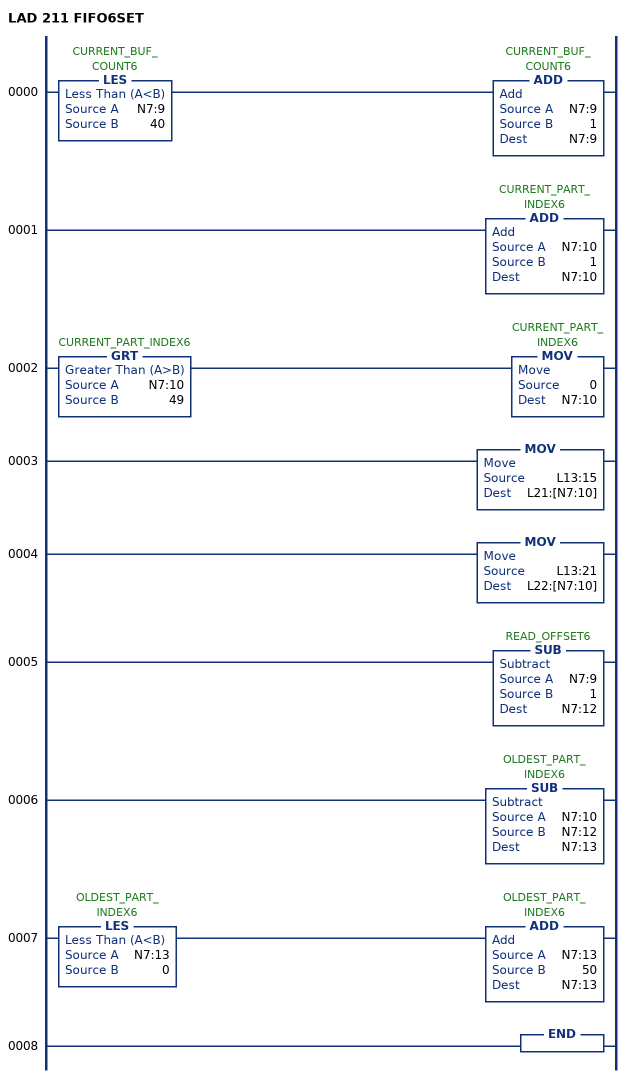
% Rung: 0 %
SOR LES N7:9 40 ADD N7:9 1 N7:9 EOR
%   N7:9  CURRENT_BUF_COUNT6 %
% Rung: 1 %
SOR ADD N7:10 1 N7:10 EOR
%   N7:10  CURRENT_PART_INDEX6 %
% Rung: 2 %
SOR GRT N7:10 49 MOV 0 N7:10 EOR
%   N7:10  CURRENT_PART_INDEX6 %
% Rung: 3 %
SOR MOV L13:15 L21:[N7:10] EOR
%   L13:15  TOP_TIME %
%   N7:10  CURRENT_PART_INDEX6 %
% Rung: 4 %
SOR MOV L13:21 L22:[N7:10] EOR
%   L13:21  TOP_POSITION %
%   N7:10  CURRENT_PART_INDEX6 %
% Rung: 5 %
SOR SUB N7:9 1 N7:12 EOR
%   N7:9  CURRENT_BUF_COUNT6 %
%   N7:12  READ_OFFSET6 %
% Rung: 6 %
SOR SUB N7:10 N7:12 N7:13 EOR
%   N7:10  CURRENT_PART_INDEX6 %
%   N7:12  READ_OFFSET6 %
%   N7:13  OLDEST_PART_INDEX6 %
% Rung: 7 %
SOR LES N7:13 0 ADD N7:13 50 N7:13 EOR
%   N7:13  OLDEST_PART_INDEX6 %
% Rung: 8 %
SOR END EOR

LADDER 212 "FIFO6GET"
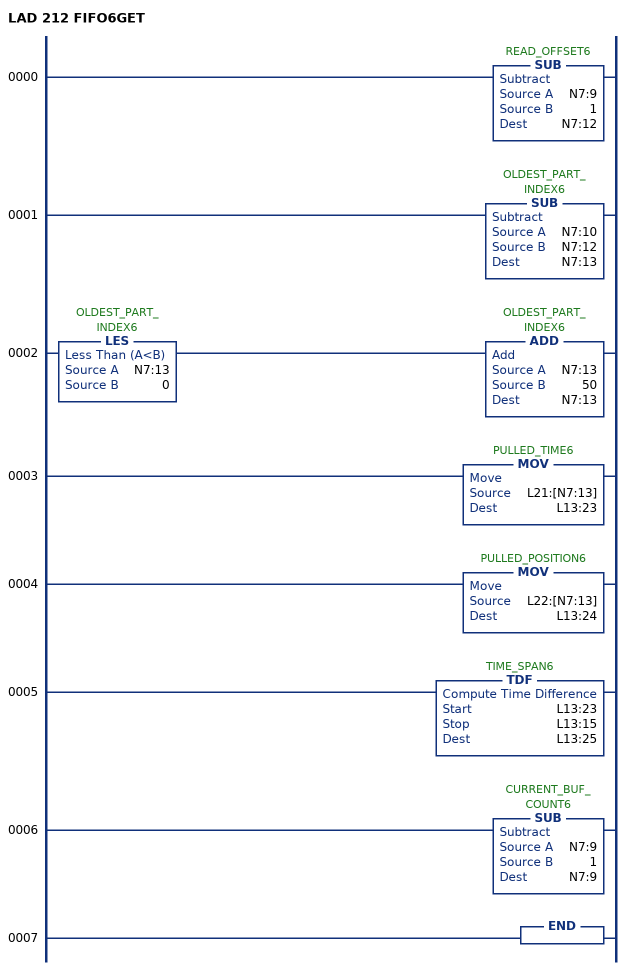
% Rung: 0 %
SOR SUB N7:9 1 N7:12 EOR
%   N7:9  CURRENT_BUF_COUNT6 %
%   N7:12  READ_OFFSET6 %
% Rung: 1 %
SOR SUB N7:10 N7:12 N7:13 EOR
%   N7:10  CURRENT_PART_INDEX6 %
%   N7:12  READ_OFFSET6 %
%   N7:13  OLDEST_PART_INDEX6 %
% Rung: 2 %
SOR LES N7:13 0 ADD N7:13 50 N7:13 EOR
%   N7:13  OLDEST_PART_INDEX6 %
% Rung: 3 %
SOR MOV L21:[N7:13] L13:23 EOR
%   N7:13  OLDEST_PART_INDEX6 %
%   L13:23  PULLED_TIME6 %
% Rung: 4 %
SOR MOV L22:[N7:13] L13:24 EOR
%   N7:13  OLDEST_PART_INDEX6 %
%   L13:24  PULLED_POSITION6 %
% Rung: 5 %
SOR TDF L13:23 L13:15 L13:25 EOR
%   L13:23  PULLED_TIME6 %
%   L13:15  TOP_TIME %
%   L13:25  TIME_SPAN6 %
% Rung: 6 %
SOR SUB N7:9 1 N7:9 EOR
%   N7:9  CURRENT_BUF_COUNT6 %
% Rung: 7 %
SOR END EOR

LADDER 213 "INSDATA6"
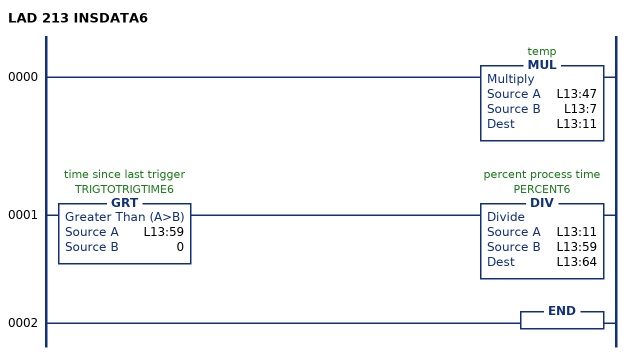
% Rung: 0 %
SOR MUL L13:47 L13:7 L13:11 EOR
%   L13:47  PROCESSTIME6  "process 6 time" %
%   L13:7  PERCENT_MULTIPLYER %
%   L13:11  "temp" %
% Rung: 1 %
SOR GRT L13:59 0 DIV L13:11 L13:59 L13:64 EOR
%   L13:59  TRIGTOTRIGTIME6  "time since last trigger" %
%   L13:11  "temp" %
%   L13:64  PERCENT6  "percent process time" %
% Rung: 2 %
SOR END EOR

LADDER 214 "TESTFAULT6"
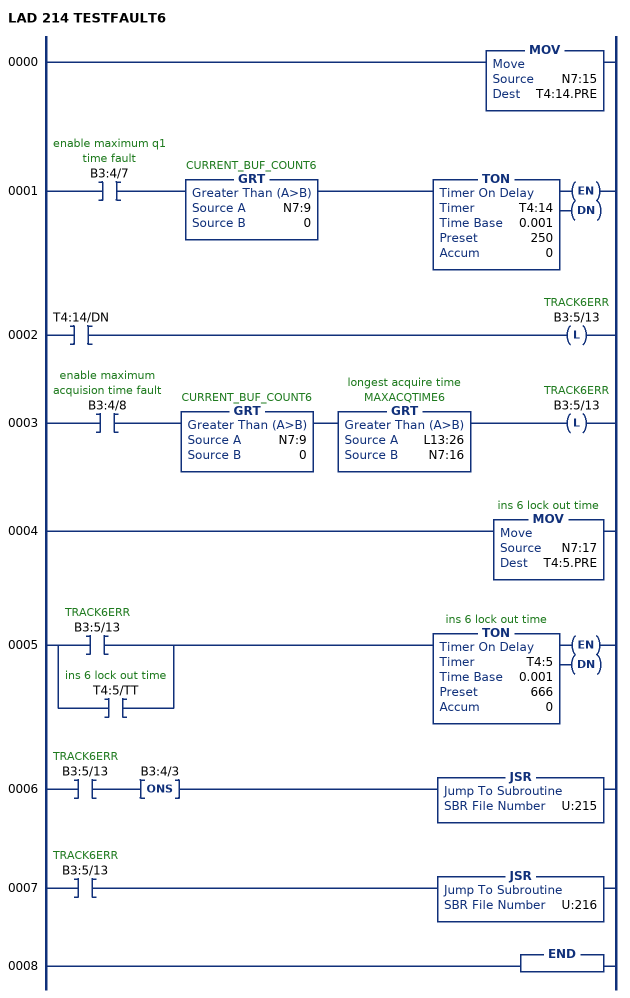
% Rung: 0 %
SOR MOV N7:15 T4:14.PRE EOR
%   N7:15  "max allowed ms time for q to be above 1 if safe fault is used" %
% Rung: 1 %
SOR XIC B3:4/7 GRT N7:9 0 TON T4:14 0.001 250 0 EOR
%   B3:4/7  "enable maximum q1 time fault" %
%   N7:9  CURRENT_BUF_COUNT6 %
% Rung: 2 %
SOR XIC T4:14/DN OTL B3:5/13 EOR
%   B3:5/13  TRACK6ERR %
% Rung: 3 %
SOR XIC B3:4/8 GRT N7:9 0 GRT L13:26 N7:16 OTL B3:5/13 EOR
%   B3:4/8  "enable maximum acquision time fault" %
%   N7:9  CURRENT_BUF_COUNT6 %
%   L13:26  MAXACQTIME6  "longest acquire time" %
%   N7:16  ACQUIRE_TIME_LIMIT  "maximum of the longest acquire time allowed if maximum acquire time fault is enabled" %
%   B3:5/13  TRACK6ERR %
% Rung: 4 %
SOR MOV N7:17 T4:5.PRE EOR
%   N7:17  "ms time setting to lock out inspection to give all pending images a chance to clear" %
%   T4:5  "ins 6 lock out time" %
% Rung: 5 %
SOR BST XIC B3:5/13 NXB XIC T4:5/TT BND TON T4:5 0.001 666 0 EOR
%   B3:5/13  TRACK6ERR %
%   T4:5  "ins 6 lock out time" %
% Rung: 6 %
SOR XIC B3:5/13 ONS B3:4/3 JSR U:215 EOR
%   B3:5/13  TRACK6ERR %
% Rung: 7 %
SOR XIC B3:5/13 JSR U:216 EOR
%   B3:5/13  TRACK6ERR %
% Rung: 8 %
SOR END EOR

LADDER 215 "INS6FIX1"
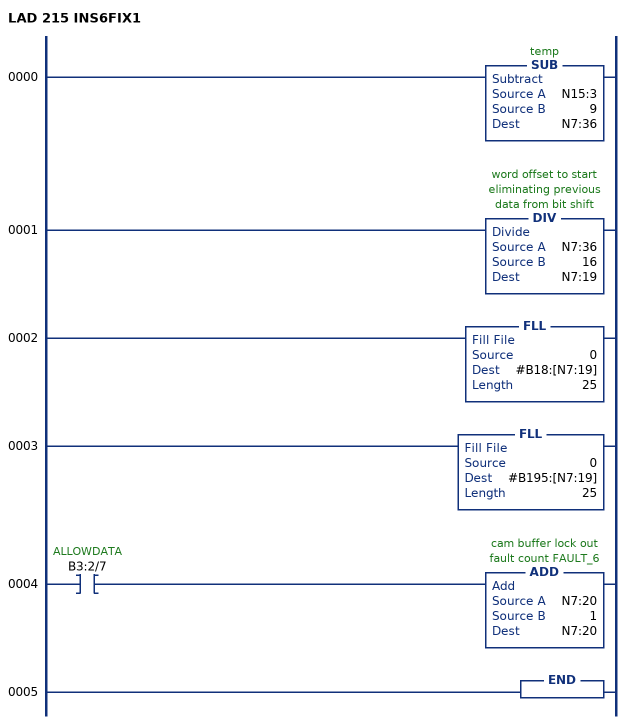
% Rung: 0 %
SOR SUB N15:3 9 N7:36 EOR
%   N15:3  INS_6_TRIG_LOC %
%   N7:36  "temp" %
% Rung: 1 %
SOR DIV N7:36 16 N7:19 EOR
%   N7:36  "temp" %
%   N7:19  "word offset to start eliminating previous data from bit shift" %
% Rung: 2 %
SOR FLL 0 #B18:[N7:19] 25 EOR
%   N7:19  "word offset to start eliminating previous data from bit shift" %
% Rung: 3 %
SOR FLL 0 #B195:[N7:19] 25 EOR
%   N7:19  "word offset to start eliminating previous data from bit shift" %
% Rung: 4 %
SOR XIC B3:2/7 ADD N7:20 1 N7:20 EOR
%   B3:2/7  ALLOWDATA %
%   N7:20  FAULT_6  "cam buffer lock out fault count" %
% Rung: 5 %
SOR END EOR

LADDER 216 "INS6FIX2"
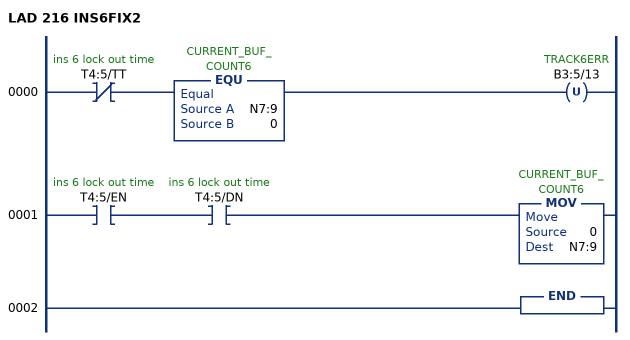
% Rung: 0 %
SOR XIO T4:5/TT EQU N7:9 0 OTU B3:5/13 EOR
%   T4:5  "ins 6 lock out time" %
%   N7:9  CURRENT_BUF_COUNT6 %
%   B3:5/13  TRACK6ERR %
% Rung: 1 %
SOR XIC T4:5/EN XIC T4:5/DN MOV 0 N7:9 EOR
%   T4:5  "ins 6 lock out time" %
%   N7:9  CURRENT_BUF_COUNT6 %
% Rung: 2 %
SOR END EOR

LADDER 218 "INS7"
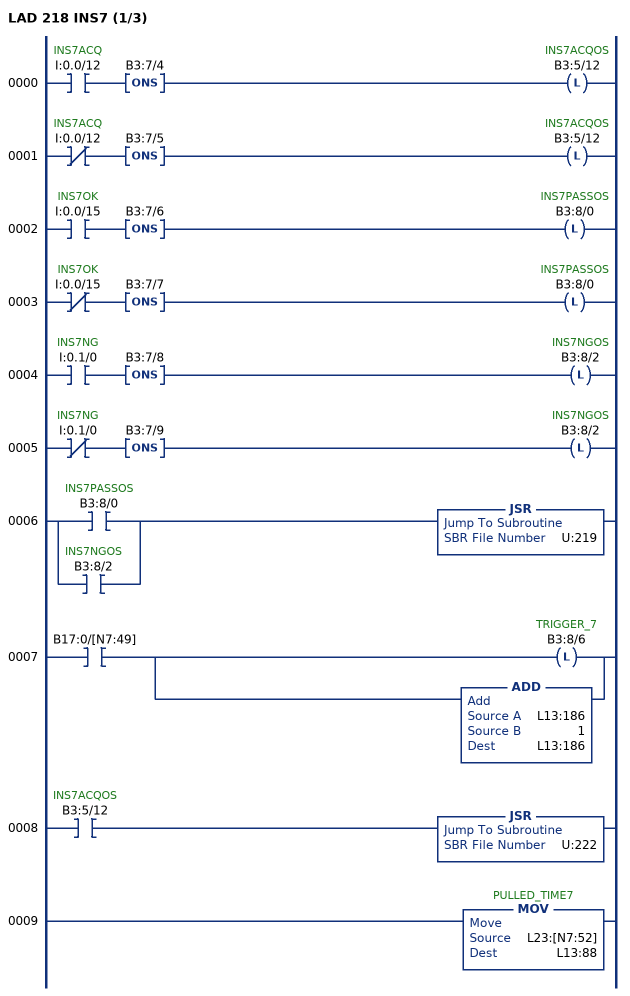
% Rung: 0 %
SOR XIC I:0.0/12 ONS B3:7/4 OTL B3:5/12 EOR
%   I:0.0/12  INS7ACQ %
%   B3:5/12  INS7ACQOS %
% Rung: 1 %
SOR XIO I:0.0/12 ONS B3:7/5 OTL B3:5/12 EOR
%   I:0.0/12  INS7ACQ %
%   B3:5/12  INS7ACQOS %
% Rung: 2 %
SOR XIC I:0.0/15 ONS B3:7/6 OTL B3:8/0 EOR
%   I:0.0/15  INS7OK %
%   B3:8/0  INS7PASSOS %
% Rung: 3 %
SOR XIO I:0.0/15 ONS B3:7/7 OTL B3:8/0 EOR
%   I:0.0/15  INS7OK %
%   B3:8/0  INS7PASSOS %
% Rung: 4 %
SOR XIC I:0.1/0 ONS B3:7/8 OTL B3:8/2 EOR
%   I:0.1/0  INS7NG %
%   B3:8/2  INS7NGOS %
% Rung: 5 %
SOR XIO I:0.1/0 ONS B3:7/9 OTL B3:8/2 EOR
%   I:0.1/0  INS7NG %
%   B3:8/2  INS7NGOS %
% Rung: 6 %
SOR BST XIC B3:8/0 NXB XIC B3:8/2 BND JSR U:219 EOR
%   B3:8/0  INS7PASSOS %
%   B3:8/2  INS7NGOS %
% Rung: 7 %
SOR XIC B17:0/[N7:49] BST OTL B3:8/6 NXB ADD L13:186 1 L13:186 BND EOR
%   B17:0  GOOD1 %
%   N7:49  INS_7_TRIG_LOC %
%   B3:8/6  TRIGGER_7 %
% Rung: 8 %
SOR XIC B3:5/12 JSR U:222 EOR
%   B3:5/12  INS7ACQOS %
% Rung: 9 %
SOR MOV L23:[N7:52] L13:88 EOR
%   N7:52  OLDEST_PART_INDEX7 %
%   L13:88  PULLED_TIME7 %

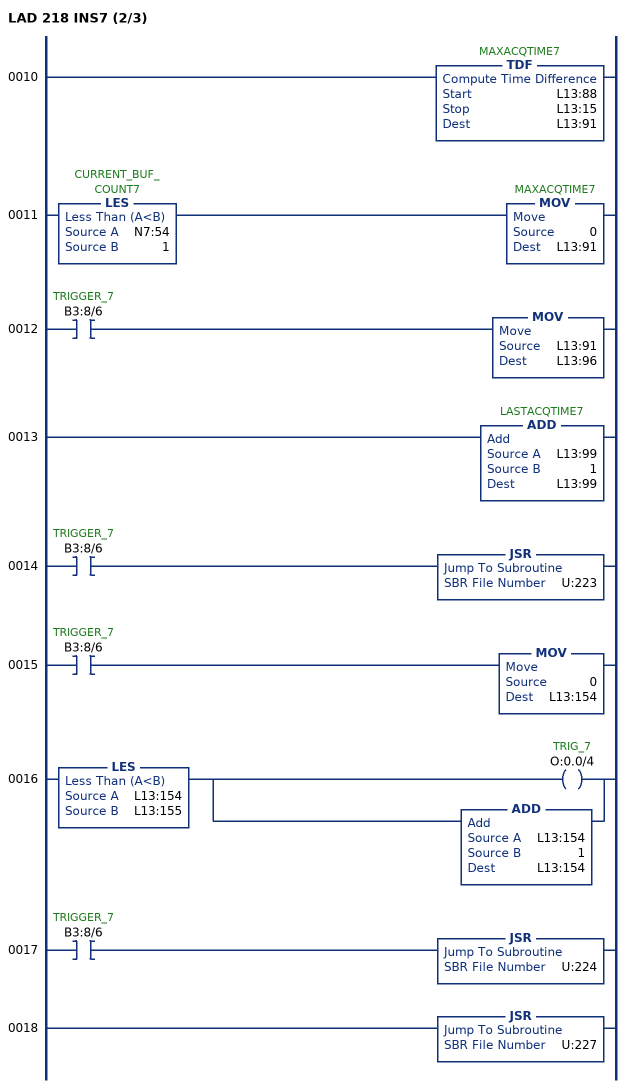
% Rung: 10 %
SOR TDF L13:88 L13:15 L13:91 EOR
%   L13:88  PULLED_TIME7 %
%   L13:15  TOP_TIME %
%   L13:91  MAXACQTIME7 %
% Rung: 11 %
SOR LES N7:54 1 MOV 0 L13:91 EOR
%   N7:54  CURRENT_BUF_COUNT7 %
%   L13:91  MAXACQTIME7 %
% Rung: 12 %
SOR XIC B3:8/6 MOV L13:91 L13:96 EOR
%   B3:8/6  TRIGGER_7 %
%   L13:91  MAXACQTIME7 %
% Rung: 13 %
SOR ADD L13:99 1 L13:99 EOR
%   L13:99  LASTACQTIME7 %
% Rung: 14 %
SOR XIC B3:8/6 JSR U:223 EOR
%   B3:8/6  TRIGGER_7 %
% Rung: 15 %
SOR XIC B3:8/6 MOV 0 L13:154 EOR
%   B3:8/6  TRIGGER_7 %
% Rung: 16 %
SOR LES L13:154 L13:155 BST OTE O:0.0/4 NXB ADD L13:154 1 L13:154 BND EOR
%   O:0.0/4  TRIG_7 %
% Rung: 17 %
SOR XIC B3:8/6 JSR U:224 EOR
%   B3:8/6  TRIGGER_7 %
% Rung: 18 %
SOR JSR U:227 EOR

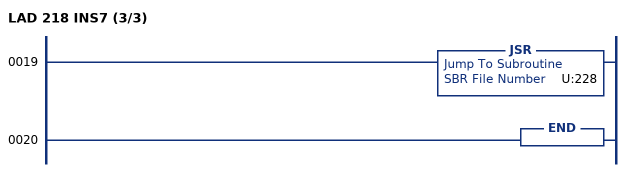
% Rung: 19 %
SOR JSR U:228 EOR
% Rung: 20 %
SOR END EOR

LADDER 219 "INS7RESULT"
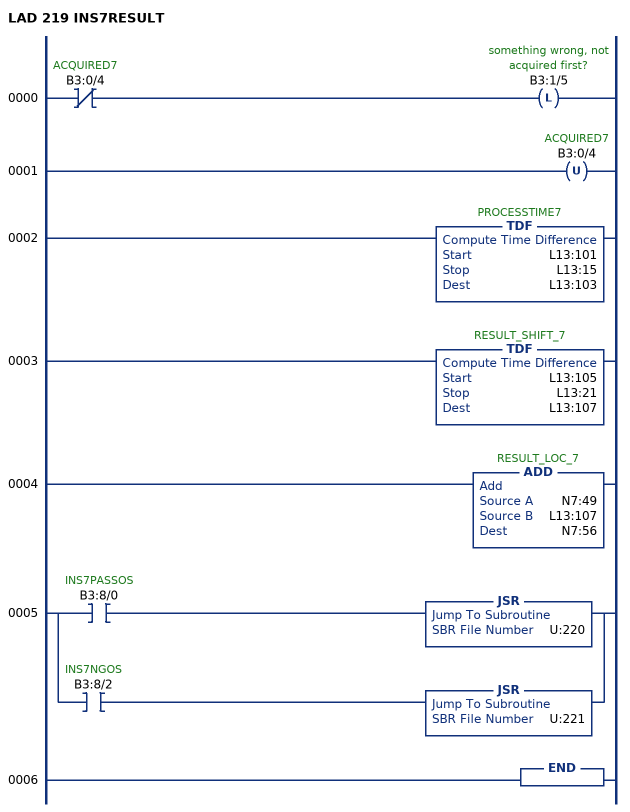
% Rung: 0 %
SOR XIO B3:0/4 OTL B3:1/5 EOR
%   B3:0/4  ACQUIRED7 %
%   B3:1/5  "something wrong, not acquired first?" %
% Rung: 1 %
SOR OTU B3:0/4 EOR
%   B3:0/4  ACQUIRED7 %
% Rung: 2 %
SOR TDF L13:101 L13:15 L13:103 EOR
%   L13:101  TIMEOFACQ7 %
%   L13:15  TOP_TIME %
%   L13:103  PROCESSTIME7 %
% Rung: 3 %
SOR TDF L13:105 L13:21 L13:107 EOR
%   L13:105  PROCESS_START_POS_7 %
%   L13:21  TOP_POSITION %
%   L13:107  RESULT_SHIFT_7 %
% Rung: 4 %
SOR ADD N7:49 L13:107 N7:56 EOR
%   N7:49  INS_7_TRIG_LOC %
%   L13:107  RESULT_SHIFT_7 %
%   N7:56  RESULT_LOC_7 %
% Rung: 5 %
SOR BST XIC B3:8/0 JSR U:220 NXB XIC B3:8/2 JSR U:221 BND EOR
%   B3:8/0  INS7PASSOS %
%   B3:8/2  INS7NGOS %
% Rung: 6 %
SOR END EOR

LADDER 220 "INS7PASS"
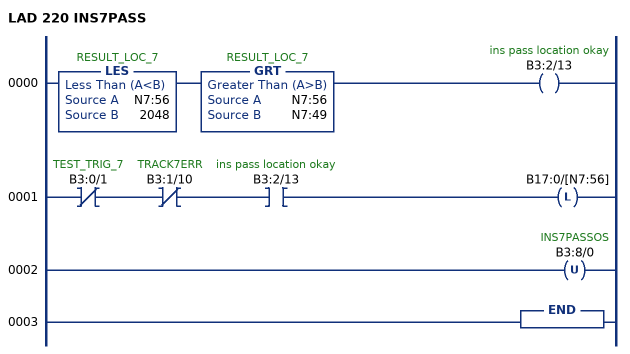
% Rung: 0 %
SOR LES N7:56 2048 GRT N7:56 N7:49 OTE B3:2/13 EOR
%   N7:56  RESULT_LOC_7 %
%   N7:49  INS_7_TRIG_LOC %
%   B3:2/13  "ins pass location okay" %
% Rung: 1 %
SOR XIO B3:0/1 XIO B3:1/10 XIC B3:2/13 OTL B17:0/[N7:56] EOR
%   B3:0/1  TEST_TRIG_7 %
%   B3:1/10  TRACK7ERR %
%   B3:2/13  "ins pass location okay" %
%   B17:0  GOOD1 %
%   N7:56  RESULT_LOC_7 %
% Rung: 2 %
SOR OTU B3:8/0 EOR
%   B3:8/0  INS7PASSOS %
% Rung: 3 %
SOR END EOR

LADDER 221 "INS7FAIL"
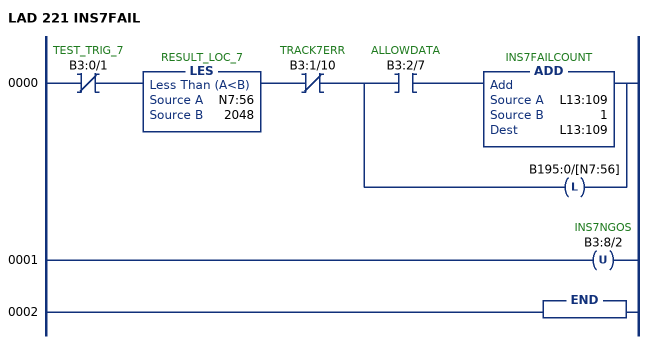
% Rung: 0 %
SOR XIO B3:0/1 LES N7:56 2048 XIO B3:1/10 BST XIC B3:2/7 ADD L13:109 1 L13:109 NXB OTL B195:0/[N7:56] BND EOR
%   B3:0/1  TEST_TRIG_7 %
%   N7:56  RESULT_LOC_7 %
%   B3:1/10  TRACK7ERR %
%   B3:2/7  ALLOWDATA %
%   L13:109  INS7FAILCOUNT %
%   B195:0  TOP_NG %
% Rung: 1 %
SOR OTU B3:8/2 EOR
%   B3:8/2  INS7NGOS %
% Rung: 2 %
SOR END EOR

LADDER 222 "INS7ACQ"
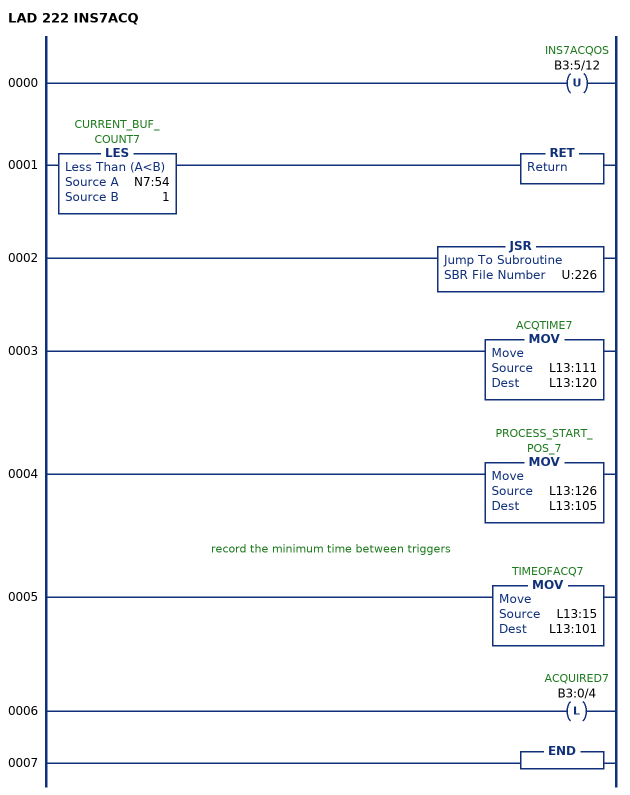
% Rung: 0 %
SOR OTU B3:5/12 EOR
%   B3:5/12  INS7ACQOS %
% Rung: 1 %
SOR LES N7:54 1 RET EOR
%   N7:54  CURRENT_BUF_COUNT7 %
% Rung: 2 %
SOR JSR U:226 EOR
% Rung: 3 %
SOR MOV L13:111 L13:120 EOR
%   L13:111  TIME_SPAN7 %
%   L13:120  ACQTIME7 %
% Rung: 4 %
SOR MOV L13:126 L13:105 EOR
%   L13:126  PULLED_POSITION7 %
%   L13:105  PROCESS_START_POS_7 %
% Rung: 5 %
% record the minimum time between triggers %
SOR MOV L13:15 L13:101 EOR
%   L13:15  TOP_TIME %
%   L13:101  TIMEOFACQ7 %
% Rung: 6 %
SOR OTL B3:0/4 EOR
%   B3:0/4  ACQUIRED7 %
% Rung: 7 %
SOR END EOR

LADDER 223 "Q7TIMETEST"
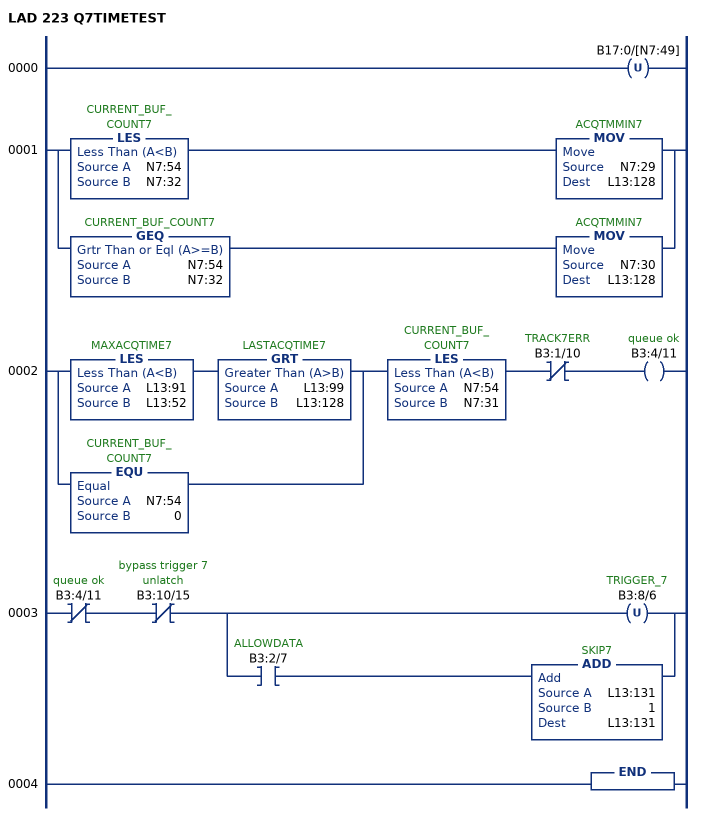
% Rung: 0 %
SOR OTU B17:0/[N7:49] EOR
%   B17:0  GOOD1 %
%   N7:49  INS_7_TRIG_LOC %
% Rung: 1 %
SOR BST LES N7:54 N7:32 MOV N7:29 L13:128 NXB GEQ N7:54 N7:32 MOV N7:30 L13:128 BND EOR
%   N7:54  CURRENT_BUF_COUNT7 %
%   N7:32  BUF_CAM_LIMIT %
%   N7:29  CAM_BUF_ACQ_TM %
%   L13:128  ACQTMMIN7 %
%   N7:30  PC_BUF_ACQ_TM %
% Rung: 2 %
SOR BST LES L13:91 L13:52 GRT L13:99 L13:128 NXB EQU N7:54 0 BND LES N7:54 N7:31 XIO B3:1/10 OTE B3:4/11 EOR
%   L13:91  MAXACQTIME7 %
%   L13:52  ACQTIMELIMIT %
%   L13:99  LASTACQTIME7 %
%   L13:128  ACQTMMIN7 %
%   N7:54  CURRENT_BUF_COUNT7 %
%   N7:31  MAX_BUFF_CT  "maximum buffers" %
%   B3:1/10  TRACK7ERR %
%   B3:4/11  "queue ok" %
% Rung: 3 %
SOR XIO B3:4/11 XIO B3:10/15 BST OTU B3:8/6 NXB XIC B3:2/7 ADD L13:131 1 L13:131 BND EOR
%   B3:4/11  "queue ok" %
%   B3:10/15  "bypass trigger 7 unlatch" %
%   B3:8/6  TRIGGER_7 %
%   B3:2/7  ALLOWDATA %
%   L13:131  SKIP7 %
% Rung: 4 %
SOR END EOR

LADDER 224 "INS7TRIG"
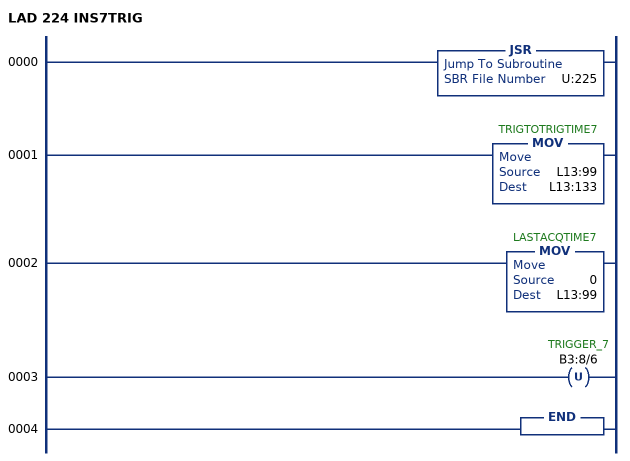
% Rung: 0 %
SOR JSR U:225 EOR
% Rung: 1 %
SOR MOV L13:99 L13:133 EOR
%   L13:99  LASTACQTIME7 %
%   L13:133  TRIGTOTRIGTIME7 %
% Rung: 2 %
SOR MOV 0 L13:99 EOR
%   L13:99  LASTACQTIME7 %
% Rung: 3 %
SOR OTU B3:8/6 EOR
%   B3:8/6  TRIGGER_7 %
% Rung: 4 %
SOR END EOR

LADDER 225 "FIFO7SET"
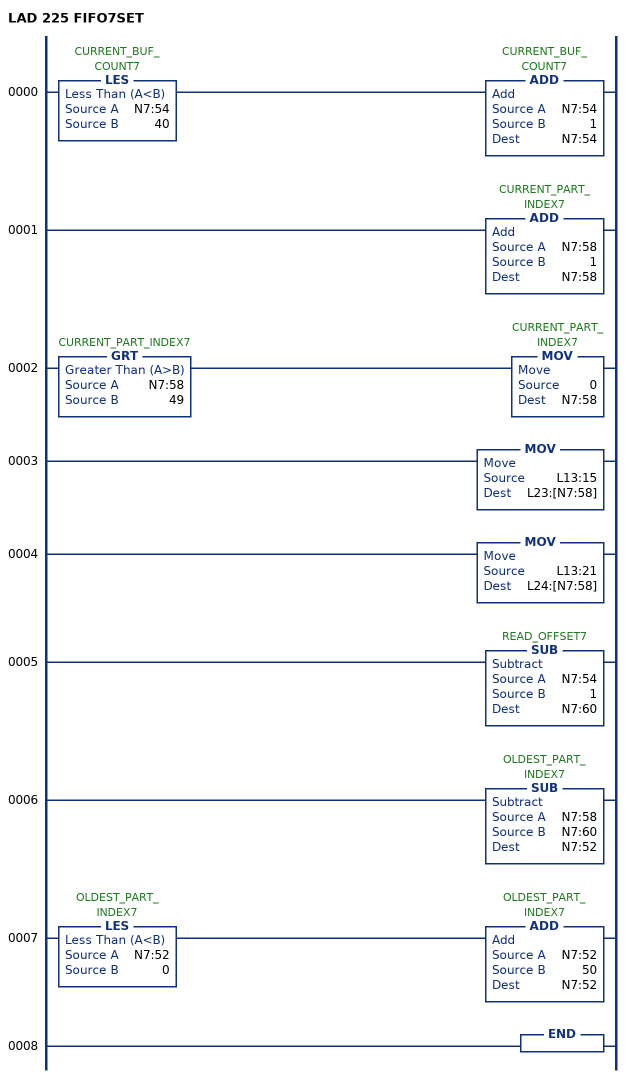
% Rung: 0 %
SOR LES N7:54 40 ADD N7:54 1 N7:54 EOR
%   N7:54  CURRENT_BUF_COUNT7 %
% Rung: 1 %
SOR ADD N7:58 1 N7:58 EOR
%   N7:58  CURRENT_PART_INDEX7 %
% Rung: 2 %
SOR GRT N7:58 49 MOV 0 N7:58 EOR
%   N7:58  CURRENT_PART_INDEX7 %
% Rung: 3 %
SOR MOV L13:15 L23:[N7:58] EOR
%   L13:15  TOP_TIME %
%   N7:58  CURRENT_PART_INDEX7 %
% Rung: 4 %
SOR MOV L13:21 L24:[N7:58] EOR
%   L13:21  TOP_POSITION %
%   N7:58  CURRENT_PART_INDEX7 %
% Rung: 5 %
SOR SUB N7:54 1 N7:60 EOR
%   N7:54  CURRENT_BUF_COUNT7 %
%   N7:60  READ_OFFSET7 %
% Rung: 6 %
SOR SUB N7:58 N7:60 N7:52 EOR
%   N7:58  CURRENT_PART_INDEX7 %
%   N7:60  READ_OFFSET7 %
%   N7:52  OLDEST_PART_INDEX7 %
% Rung: 7 %
SOR LES N7:52 0 ADD N7:52 50 N7:52 EOR
%   N7:52  OLDEST_PART_INDEX7 %
% Rung: 8 %
SOR END EOR

LADDER 226 "FIFO7GET"
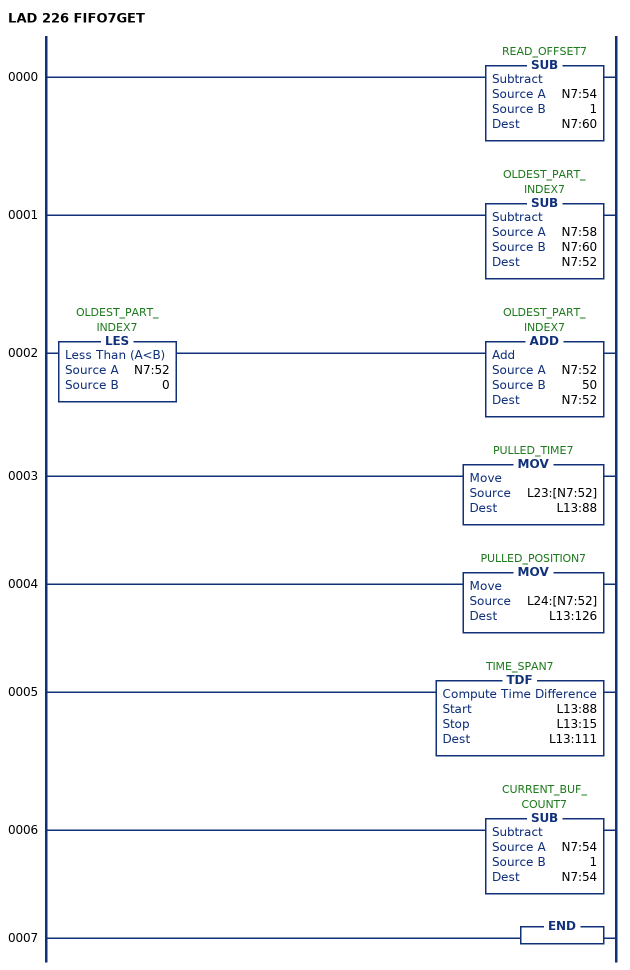
% Rung: 0 %
SOR SUB N7:54 1 N7:60 EOR
%   N7:54  CURRENT_BUF_COUNT7 %
%   N7:60  READ_OFFSET7 %
% Rung: 1 %
SOR SUB N7:58 N7:60 N7:52 EOR
%   N7:58  CURRENT_PART_INDEX7 %
%   N7:60  READ_OFFSET7 %
%   N7:52  OLDEST_PART_INDEX7 %
% Rung: 2 %
SOR LES N7:52 0 ADD N7:52 50 N7:52 EOR
%   N7:52  OLDEST_PART_INDEX7 %
% Rung: 3 %
SOR MOV L23:[N7:52] L13:88 EOR
%   N7:52  OLDEST_PART_INDEX7 %
%   L13:88  PULLED_TIME7 %
% Rung: 4 %
SOR MOV L24:[N7:52] L13:126 EOR
%   N7:52  OLDEST_PART_INDEX7 %
%   L13:126  PULLED_POSITION7 %
% Rung: 5 %
SOR TDF L13:88 L13:15 L13:111 EOR
%   L13:88  PULLED_TIME7 %
%   L13:15  TOP_TIME %
%   L13:111  TIME_SPAN7 %
% Rung: 6 %
SOR SUB N7:54 1 N7:54 EOR
%   N7:54  CURRENT_BUF_COUNT7 %
% Rung: 7 %
SOR END EOR

LADDER 227 "INSDATA7"
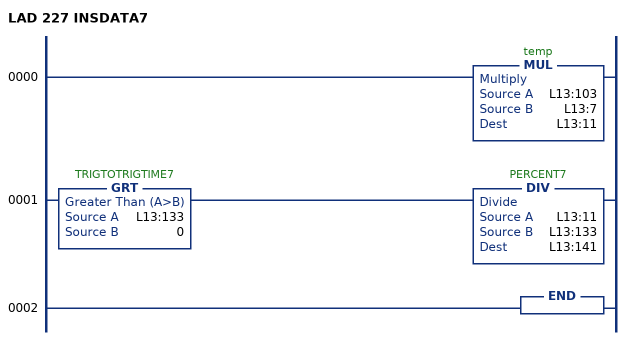
% Rung: 0 %
SOR MUL L13:103 L13:7 L13:11 EOR
%   L13:103  PROCESSTIME7 %
%   L13:7  PERCENT_MULTIPLYER %
%   L13:11  "temp" %
% Rung: 1 %
SOR GRT L13:133 0 DIV L13:11 L13:133 L13:141 EOR
%   L13:133  TRIGTOTRIGTIME7 %
%   L13:11  "temp" %
%   L13:141  PERCENT7 %
% Rung: 2 %
SOR END EOR

LADDER 228 "TESTFAULT7"
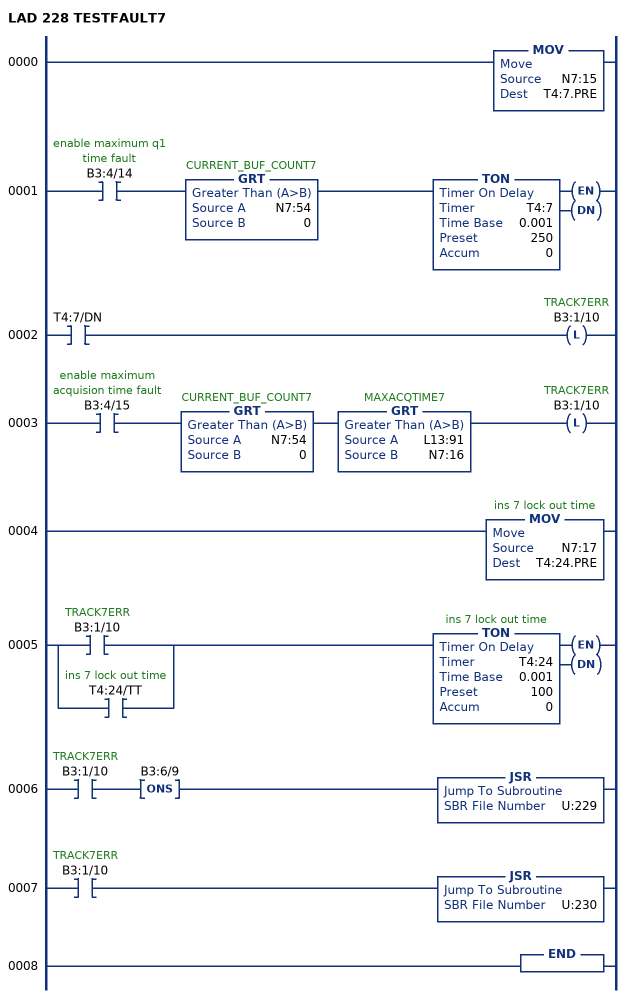
% Rung: 0 %
SOR MOV N7:15 T4:7.PRE EOR
%   N7:15  "max allowed ms time for q to be above 1 if safe fault is used" %
% Rung: 1 %
SOR XIC B3:4/14 GRT N7:54 0 TON T4:7 0.001 250 0 EOR
%   B3:4/14  "enable maximum q1 time fault" %
%   N7:54  CURRENT_BUF_COUNT7 %
% Rung: 2 %
SOR XIC T4:7/DN OTL B3:1/10 EOR
%   B3:1/10  TRACK7ERR %
% Rung: 3 %
SOR XIC B3:4/15 GRT N7:54 0 GRT L13:91 N7:16 OTL B3:1/10 EOR
%   B3:4/15  "enable maximum acquision time fault" %
%   N7:54  CURRENT_BUF_COUNT7 %
%   L13:91  MAXACQTIME7 %
%   N7:16  ACQUIRE_TIME_LIMIT  "maximum of the longest acquire time allowed if maximum acquire time fault is enabled" %
%   B3:1/10  TRACK7ERR %
% Rung: 4 %
SOR MOV N7:17 T4:24.PRE EOR
%   N7:17  "ms time setting to lock out inspection to give all pending images a chance to clear" %
%   T4:24  "ins 7 lock out time" %
% Rung: 5 %
SOR BST XIC B3:1/10 NXB XIC T4:24/TT BND TON T4:24 0.001 100 0 EOR
%   B3:1/10  TRACK7ERR %
%   T4:24  "ins 7 lock out time" %
% Rung: 6 %
SOR XIC B3:1/10 ONS B3:6/9 JSR U:229 EOR
%   B3:1/10  TRACK7ERR %
% Rung: 7 %
SOR XIC B3:1/10 JSR U:230 EOR
%   B3:1/10  TRACK7ERR %
% Rung: 8 %
SOR END EOR

LADDER 229 "INS7FIX1"
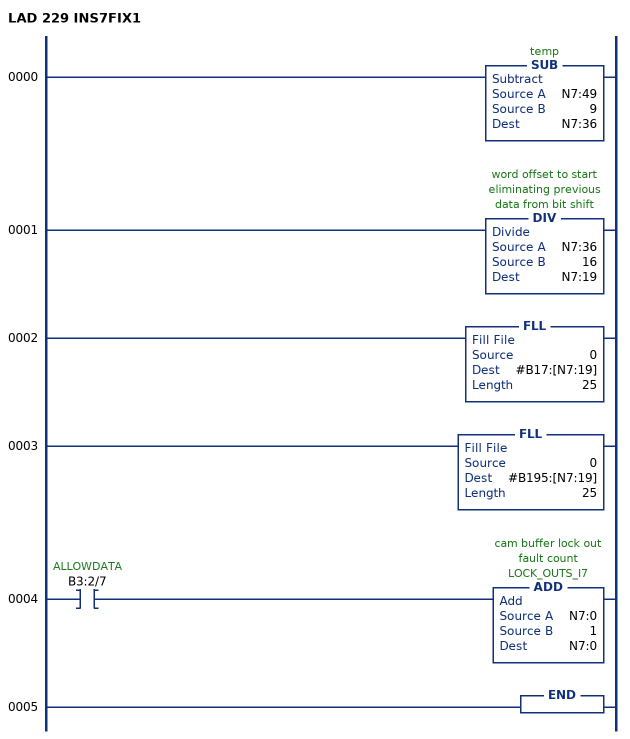
% Rung: 0 %
SOR SUB N7:49 9 N7:36 EOR
%   N7:49  INS_7_TRIG_LOC %
%   N7:36  "temp" %
% Rung: 1 %
SOR DIV N7:36 16 N7:19 EOR
%   N7:36  "temp" %
%   N7:19  "word offset to start eliminating previous data from bit shift" %
% Rung: 2 %
SOR FLL 0 #B17:[N7:19] 25 EOR
%   N7:19  "word offset to start eliminating previous data from bit shift" %
% Rung: 3 %
SOR FLL 0 #B195:[N7:19] 25 EOR
%   N7:19  "word offset to start eliminating previous data from bit shift" %
% Rung: 4 %
SOR XIC B3:2/7 ADD N7:0 1 N7:0 EOR
%   B3:2/7  ALLOWDATA %
%   N7:0  LOCK_OUTS_I7  "cam buffer lock out fault count" %
% Rung: 5 %
SOR END EOR

LADDER 230 "INS7FIX2"
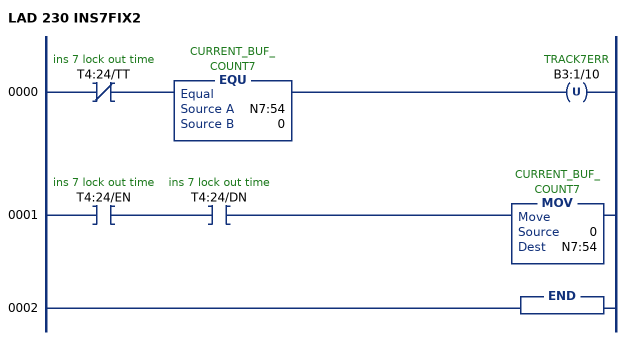
% Rung: 0 %
SOR XIO T4:24/TT EQU N7:54 0 OTU B3:1/10 EOR
%   T4:24  "ins 7 lock out time" %
%   N7:54  CURRENT_BUF_COUNT7 %
%   B3:1/10  TRACK7ERR %
% Rung: 1 %
SOR XIC T4:24/EN XIC T4:24/DN MOV 0 N7:54 EOR
%   T4:24  "ins 7 lock out time" %
%   N7:54  CURRENT_BUF_COUNT7 %
% Rung: 2 %
SOR END EOR

LADDER 232 "INS8"
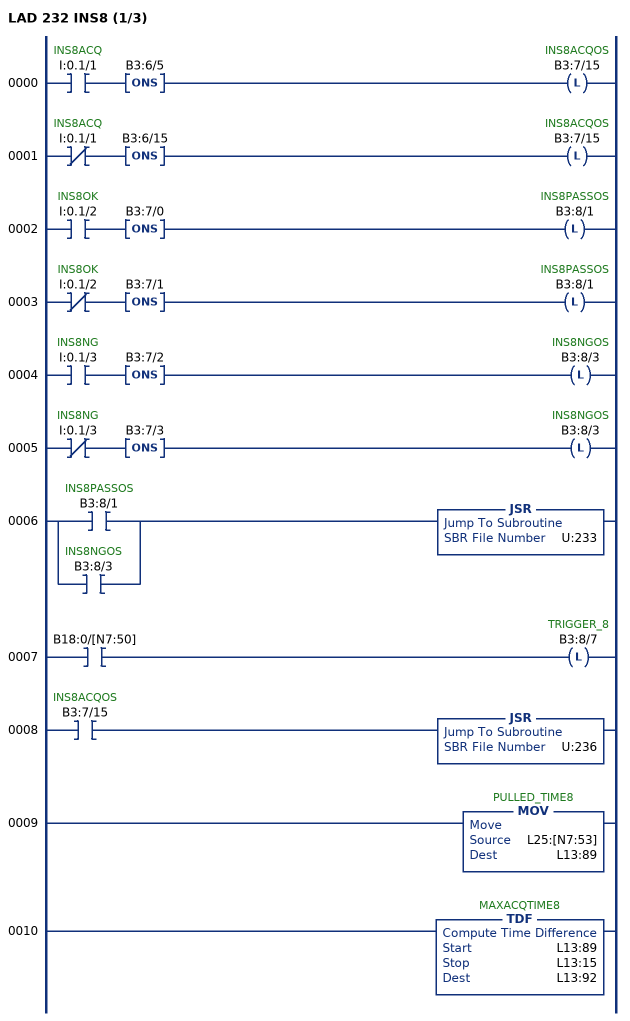
% Rung: 0 %
SOR XIC I:0.1/1 ONS B3:6/5 OTL B3:7/15 EOR
%   I:0.1/1  INS8ACQ %
%   B3:7/15  INS8ACQOS %
% Rung: 1 %
SOR XIO I:0.1/1 ONS B3:6/15 OTL B3:7/15 EOR
%   I:0.1/1  INS8ACQ %
%   B3:7/15  INS8ACQOS %
% Rung: 2 %
SOR XIC I:0.1/2 ONS B3:7/0 OTL B3:8/1 EOR
%   I:0.1/2  INS8OK %
%   B3:8/1  INS8PASSOS %
% Rung: 3 %
SOR XIO I:0.1/2 ONS B3:7/1 OTL B3:8/1 EOR
%   I:0.1/2  INS8OK %
%   B3:8/1  INS8PASSOS %
% Rung: 4 %
SOR XIC I:0.1/3 ONS B3:7/2 OTL B3:8/3 EOR
%   I:0.1/3  INS8NG %
%   B3:8/3  INS8NGOS %
% Rung: 5 %
SOR XIO I:0.1/3 ONS B3:7/3 OTL B3:8/3 EOR
%   I:0.1/3  INS8NG %
%   B3:8/3  INS8NGOS %
% Rung: 6 %
SOR BST XIC B3:8/1 NXB XIC B3:8/3 BND JSR U:233 EOR
%   B3:8/1  INS8PASSOS %
%   B3:8/3  INS8NGOS %
% Rung: 7 %
SOR XIC B18:0/[N7:50] OTL B3:8/7 EOR
%   B18:0  GOOD2 %
%   N7:50  INS_8_TRIG_LOC %
%   B3:8/7  TRIGGER_8 %
% Rung: 8 %
SOR XIC B3:7/15 JSR U:236 EOR
%   B3:7/15  INS8ACQOS %
% Rung: 9 %
SOR MOV L25:[N7:53] L13:89 EOR
%   N7:53  OLDEST_PART_INDEX8 %
%   L13:89  PULLED_TIME8 %
% Rung: 10 %
SOR TDF L13:89 L13:15 L13:92 EOR
%   L13:89  PULLED_TIME8 %
%   L13:15  TOP_TIME %
%   L13:92  MAXACQTIME8 %

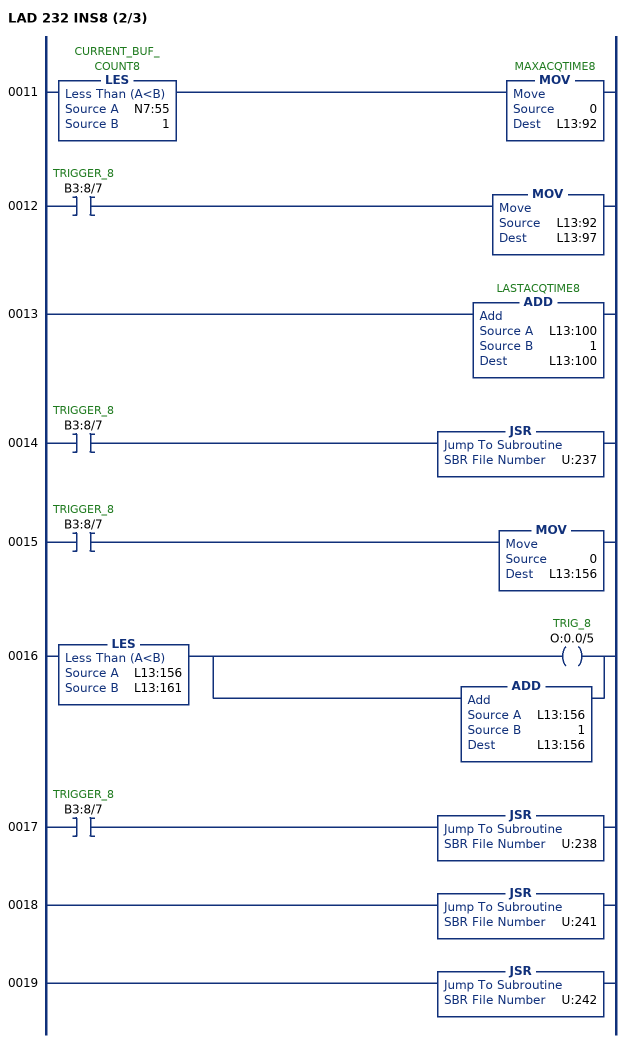
% Rung: 11 %
SOR LES N7:55 1 MOV 0 L13:92 EOR
%   N7:55  CURRENT_BUF_COUNT8 %
%   L13:92  MAXACQTIME8 %
% Rung: 12 %
SOR XIC B3:8/7 MOV L13:92 L13:97 EOR
%   B3:8/7  TRIGGER_8 %
%   L13:92  MAXACQTIME8 %
% Rung: 13 %
SOR ADD L13:100 1 L13:100 EOR
%   L13:100  LASTACQTIME8 %
% Rung: 14 %
SOR XIC B3:8/7 JSR U:237 EOR
%   B3:8/7  TRIGGER_8 %
% Rung: 15 %
SOR XIC B3:8/7 MOV 0 L13:156 EOR
%   B3:8/7  TRIGGER_8 %
% Rung: 16 %
SOR LES L13:156 L13:161 BST OTE O:0.0/5 NXB ADD L13:156 1 L13:156 BND EOR
%   O:0.0/5  TRIG_8 %
% Rung: 17 %
SOR XIC B3:8/7 JSR U:238 EOR
%   B3:8/7  TRIGGER_8 %
% Rung: 18 %
SOR JSR U:241 EOR
% Rung: 19 %
SOR JSR U:242 EOR

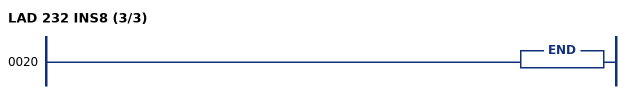
% Rung: 20 %
SOR END EOR

LADDER 233 "INS8RESULT"
